(* PLC project Generated.project, CODESYS CODESYS V3.5 SP19 Patch 1 *)
(* stored: creationDateTime 2026-08-11T14:02:33.684370, modificationDateTime 2026-08-11T14:02:33.684370 *)

(* ═══════════════════════════════════════════════════════════════ ↔️ ST_TranslationHMI — Données d'échange IHM pour le Translation M3 ─────────────────────────────────────────────────────────────── 🎨 Destiné à l'affichage des états, commandes et diagnostics du translation. 📄 Structuration en Cmd / State / Safety / Bypass / Test (2026-07-22) — doc métier : ARCHIVES/Doc/AF_Partie-11_Fonction_Translation_v2.0.md ═══════════════════════════════════════════════════════════════ *)
TYPE ST_TranslationHMI : STRUCT
  Cmd : ST_TranslationCmd;  (* 🎮 Commandes opérateur (manuel / maintenance) *)
  State : ST_TranslationState;  (* 🚦 États & diagnostics *)
  Cfg : ST_TranslationCfg;  (* 🔧 Configurations et limites — 🆕 2026-08-06, manquait (contrairement à ST_WinchHMI) *)
  Bypass : ST_BypassTranslation;  (* 🔧 Bypass maintenance *)
  Safety : ST_SafetyTranslation;  (* 🛡️ Sécurité (FB_Safety_Translation) *)
END_STRUCT;
END_TYPE

(* ═══════════════════════════════════════════════════════════════ 🔧 ST_BypassTranslation — Bypass maintenance dédiés à Translation M3 ─────────────────────────────────────────────────────────────── 🔒 Doctrine : actionnable UNIQUEMENT en MAINT_N2, RETAIN, jamais masque les autres défauts du même bloc (voir REGISTRE_ACTIONS_Bypass_v1.0 (archive)). ═══════════════════════════════════════════════════════════════ *)
TYPE ST_BypassTranslation : STRUCT
  OperatorComm : BOOL;  (* 📡 1. Communication & Systèmes auxiliaires 📡 Bypass communication esclave CANopen Joystick / heartbeat IHM *)
  DriveComm : BOOL;  (* 📡 Bypass diagnostic esclave EtherCAT AC600 (variateur) *)
  ContactorFeedback : BOOL;  (* 🔌 Bypass feedbacks contacteur de frein *)
  PhaseRotation : BOOL;  (* ⚡ Bypass défaut rotation de phases (commun machine) *)
  BrakeThermal : BOOL;  (* 🌡️ Bypass surchauffe thermique frein (commun machine) *)
  LimitSwitch : BOOL;  (* 🚧 2. Limites physiques et Positionnement 🚧 Bypass fins de course physiques avant/arrière *)
  SensorIncoherent : BOOL;  (* 🧭 Bypass incohérence mot capteurs de position *)
  MinHeight : BOOL;  (* 🆕 2026-08-06 : Bypass interlock hauteur mini M1/M2 requise pour translation *)
  MecaA : BOOL;  (* ⚙️ 3. Sécurité Mécanique (Méca A-B) 🔄 Bypass Méca A : mouvement non commandé à l'arrêt *)
  MecaB : BOOL;  (* 🛑 Bypass Méca B : absence confirmation arrêt (frein/contacteurs) *)
  Safety : BOOL;  (* 🛡️ 4. Hiérarchie & Restauration 🛡️ Bypass groupé : tous les bits qui provoquent un PowerCutOff *)
  Process : BOOL;  (* ⚙️ Bypass groupé : tous les bits qui provoquent un SafeStop *)
  Global : BOOL;  (* 🌐 Bypass Global : ignore toutes les sécurités de cet axe *)
  Initialized : BOOL := FALSE;  (* 🐛 FIX persistance (voir DOC/AUDITS/ConfigPersistence/) : flag restauration boot dédié (défaut FALSE non ambigu, contrairement à une valeur métier) — PRG_SUPERVISION_CFC.st 🚦 TRUE = bypass restauré depuis GVL_BypassRetain ce boot *)
END_STRUCT;
END_TYPE

(* ═══════════════════════════════════════════════════════════════ 🛡️ ST_SafetyTranslation — Diagnostics de sécurité pour la Translation M3 ─────────────────────────────────────────────────────────────── 🎨 Destiné à l'affichage des défauts de sécurité du translation. ═══════════════════════════════════════════════════════════════ *)
TYPE ST_SafetyTranslation : STRUCT
  Error : BOOL;  (* 🛡️ Bloc sécurité (Safety) en défaut *)
  ErrorId : WORD;  (* ❌ Code bitfield du défaut de sécurité *)
  ErrorOperatorComm : BOOL;  (* 🎮 Perte communication opérateur : joystick CAN ou heartbeat IHM (bit0) *)
  ErrorDriveComm : BOOL;  (* 📡 Perte communication EtherCAT variateur (bit1) *)
  ErrorPhaseRotation : BOOL;  (* ⚡ Mauvaise rotation de phases électriques (bit2) *)
  ErrorBrakeThermal : BOOL;  (* 🌡️ Surchauffe thermique frein commun (bit3) *)
  ErrorMecaB : BOOL;  (* 🛑 Absence confirmation arrêt (Méca B - bit4) *)
  ErrorMecaA : BOOL;  (* 🔄 Mouvement non commandé (Méca A - bit5) *)
  ErrorLimitSwitch : BOOL;  (* 🚧 Limite extrême Translation atteinte (bit6) *)
  ErrorSensorIncoherent : BOOL;  (* 🧭 Mot capteurs M3 incohérent (bit7) *)
  SafeStop : BOOL;  (* 🛡️ Décélération de sécurité demandée *)
  PowerCutOff : BOOL;  (* 🧨 Coupure puissance demandée *)
END_STRUCT;
END_TYPE

(* ═══════════════════════════════════════════════════════════════ 🔧 ST_TranslationCfg — Configurations et paramètres réglables pour Translation M3 ─────────────────────────────────────────────────────────────── 🎨 Destiné au paramétrage depuis l'IHM (RETAIN) — même patron que ST_WinchCfg. 📄 2026-08-06 : créé suite constat terrain — Translation n'avait pas de slot Cfg (contrairement à ST_WinchHMI), les 3 vitesses de ralentissement d'approche n'étaient donc réglables qu'en dur dans GVL_PERSISTENT (recompilation requise). ═══════════════════════════════════════════════════════════════ *)
TYPE ST_TranslationCfg : STRUCT
  CfgApproachSpeedTremie_Hz : REAL := 10;  (* 🐢 Vitesse réduite d'approche Trémie (Hz), déclenchée par capteur PV, Direction=1 *)
  CfgApproachSpeedMaintenance_Hz : REAL := 10;  (* 🐢 Vitesse réduite d'approche Maintenance (Hz), déclenchée par capteur P1, Direction=-1 *)
  CfgApproachSpeedP1_Hz : REAL := 10;  (* 🐢 Vitesse réduite d'approche P1 (Hz), déclenchée par capteur P2, Direction=-1 *)
  Initialized : BOOL := FALSE;  (* 🐛 Flag restauration boot (défaut FALSE non ambigu) — même patron que ST_WinchCfg 🚦 TRUE = config restaurée depuis GVL_PERSISTENT ce boot *)
END_STRUCT;
END_TYPE

(* ═══════════════════════════════════════════════════════════════ 🎮 ST_TranslationCmd — Commandes IHM pour la Translation M3 ─────────────────────────────────────────────────────────────── 🎨 Destiné au pilotage de la translation M3 depuis l'IHM. 📄 2026-07-24 : Initialized protège SetFreq_Hz (seul réglage à survivre au reboot), sans pont générique pour ne jamais persister BtnFwd/BtnRev. ═══════════════════════════════════════════════════════════════ *)
TYPE ST_TranslationCmd : STRUCT
  SelPositioning : BOOL;  (* 🎯 TRUE = positionneur sur SelTarget ; FALSE = jog libre *)
  SelTarget : INT;  (* 🔢 Numéro de la cible de position sélectionnée *)
  BtnFwd : BOOL;  (* ↔️ Requête marche avant (→ Trémie), pilotage IHM exclusif *)
  BtnRev : BOOL;  (* ↔️ Requête marche arrière (→ Maintenance), pilotage IHM exclusif *)
  SetFreq_Hz : REAL;  (* 🎯 Consigne fréquence manuelle [Hz], limitée par PRG_10_Outputs_LD *)
  InvertDirection : BOOL;  (* 🔀 2026-08-06 : TglJoystickMaster PAR AXE supprimé (doublon) — un seul switch machine : GVL_IHM.Modes.Cmd.TglJoystickMaster (ST_ModesCmd), applicable à M1/M2 ET M3. 🔄 TRUE = inverse Fwd→Maintenance / Rev→Trémie (mise en service) *)
  TglMaintenanceZoneAccess : BOOL;  (* 🆕 2026-08-06 : autorisation CONSCIENTE zone Maintenance, EN PLUS de MAINT_N2 (Auth.MaintenanceM3TargetEnable) *)
  Initialized : BOOL := FALSE;  (* 🚦 TRUE = SetFreq_Hz restauré depuis GVL_PERSISTENT ce boot *)
END_STRUCT;
END_TYPE

(* ═══════════════════════════════════════════════════════════════ 🚦 ST_TranslationState — États et retours IHM pour la Translation M3 ─────────────────────────────────────────────────────────────── 🎨 Destiné à l'affichage des retours et mesures de la translation M3. ═══════════════════════════════════════════════════════════════ *)
TYPE ST_TranslationState : STRUCT
  FBState : E_State;  (* 🚦 États & diagnostics FB_Translation 🤖 État de l'automate interne (FB_Translation) *)
  Ready : BOOL;  (* 🟢 Translation prêt à fonctionner *)
  Busy : BOOL;  (* ⚙️ Mouvement en cours *)
  Done : BOOL;  (* ✅ Mouvement terminé avec succès *)
  Error : BOOL;  (* 🔴 Translation en défaut *)
  ErrorId : WORD;  (* ❌ Code du défaut actif *)
  BrakeCmd : BOOL;  (* 🔓 Commande de desserrage du frein (lecture seule, TRUE = desserré) *)
  BrakeFeedback : BOOL;  (* 🔌 Retour physique direct : TRUE = frein OUVERT (desserré) *)
  PositionSensorTarget : BOOL;  (* 🎯 Capteur de détection de la position cible atteint *)
  PositionReached : BOOL;  (* ✅ Positionneur : cible sélectionnée atteinte (non mémorisé) *)
  JoystickDeflection_Pct : REAL;  (* 🕹️ Axe X fonctionnel -100..+100 %, 0 = neutre ; animation IHM M3 *)
  DriveActualFreq_Hz : REAL;  (* 📈 Fréquence de sortie réelle du variateur (Hz) *)
  DriveControlWord : WORD;  (* ⚙️ Mot de commande AC600 réellement appliqué *)
  DriveFreqRef_Hz : REAL;  (* 🎯 Consigne fréquence réellement appliquée *)
  ActiveDirection : INT;  (* ↔️ Sens arbitré : -1 / 0 / +1 *)
  ActiveSpeedRef_Pct : REAL;  (* 📊 Consigne active après arbitrage *)
  FinalInterlockState : E_State;  (* 🛡️ État final _LD lecture seule *)
  FinalInterlockReason : E_TranslationFinalInterlockReason;  (* 🛡️ Cause finale mémorisée *)
  FinalInterlockError : BOOL;  (* 🛡️ Défaut final mémorisé *)
  FinalInterlockErrorId : WORD;  (* 🛡️ Bitfield final *)
  BrakeCommandOpenConfirmed : BOOL;  (* 🔌 Contacteur/bobine desserrage confirmé, pas frein mécanique *)
  FinalBrakeTimeoutElapsed : TIME;  (* ⏱️ Écoulé watchdog 500ms *)
  DriveCommReady : BOOL;  (* 🔌 Diagnostic variateur EtherCAT (décodé — pas de bit-masking côté IHM) 📡 Variateur M3 : communication prête (StatusWord bit7) *)
  DrivePowerReady : BOOL;  (* ⚡ Variateur M3 : puissance prête (StatusWord bit0) *)
  PositionTremie : BOOL;  (* 📍 Mot capteurs et positions Translation M3 *)
  PositionPV : BOOL;
  PositionP2 : BOOL;
  PositionP1 : BOOL;
  PositionMaintenance : BOOL;
  AtTremie : BOOL;  (* 🆕 2026-08-06 : mot EXACT — front franc arrivée/cible (voir PositionXxx ci-dessus = cumulatif zone, réservé ralentissement) *)
  AtPV : BOOL;
  AtP2 : BOOL;
  AtP1 : BOOL;
  AtMaintenance : BOOL;
  EstimatedPosM3_M : REAL;  (* 📏 Position continue estimée en mètres (0.0 m Maint -> +X m Trémie) — persistante, survit reboot *)
  SensorsWord : BYTE;  (* bit4=Trémie, bit3=PV, bit2=P2, bit1=P1, bit0=Maintenance *)
  SensorWordIncoherent : BOOL;
  LimitSwitchFwd : BOOL;
  LimitSwitchRev : BOOL;
  DriveThermalOk : BOOL;  (* 🆕 T96 : retour disjoncteur thermique moteur/variateur AC600 — diagnostic seul, l'AC600 se protège déjà lui-même *)
  MaintenanceTargetEnable : BOOL;  (* 🔓 TRUE = Autorise le déplacement vers la cible 4 (Maintenance) ; actif uniquement en mode MAINT_N2 *)
  SimulationModeActive : BOOL;
  HeightInterlockBlocking : BOOL;  (* 🆕 2026-08-06 : TRUE = translation bloquée, M1 ou M2 sous la hauteur mini requise *)
END_STRUCT;
END_TYPE

(* values of E_State: DISABLED: Enable faux, neutralisé; INIT: Démarrage / vérifs; READY: Prêt, attend ordre; BUSY: Action en cours; DONE: Action terminée; STOPPING: Décél rampe avant arrêt (StartStop=FALSE ou SafeStop=TRUE) *)

{attribute 'qualified_only'}
{attribute 'strict'}
TYPE E_State : (DISABLED := 0, INIT := 1, READY := 2, BUSY := 3, DONE := 4, STOPPING := 5);
END_TYPE

{attribute 'qualified_only'}
{attribute 'strict'}
TYPE E_TranslationFinalInterlockReason : (NONE := 0, BRAKE_COMMAND_NOT_CONFIRMED := 1, RESTART_INHIBITED := 2);
END_TYPE
